FUNCTION_BLOCK BurnOffStation
VAR_INPUT
END_VAR
VAR_OUTPUT
END_VAR
VAR
	HeaterONTimer : TON;
	BlowerOFFTimer : TON;
	PrevRunning, CurrRunning : BOOL := FALSE;
	StartFromReset, StopAfterEStop : BOOL:=FALSE;	
	BlowerEnable: BOOL := FALSE;
	HeatEnable: BOOL := FALSE;
	PIDEnable: BOOL := FALSE;
	nErrorPIDStatus : UINT;
	PIDOutput : LREAL;
	VoltOutReal : LREAL;
	fbBurnoffPID :FB_BasicPID;
	// Temperature needs to be divided by 10 after reading from the TC card
	fProcessValue: LREAL := 0;
END_VAR

fProcessValue := GVL_IO.BU_Temperature/10;	
STATUS.BurnOffTemperature := LREAL_TO_DINT(fProcessValue);

IF (NOT LotsData.Lot.BurnOffEnabled OR STATIONS.fbMMMonitor.IsMMJammed OR Stations.fbCycleControl.StopRequested OR GVL_IO.MachineEStopped OR Status.BurnOffIdle) THEN
	GVL_IO.BU_HeatCntl := 0;
	GVL_IO.BU_BlowCntl := 0;
ELSE 
	// set the blower setpoint from the User configuration in HMI
	GVL_IO.BU_BlowCntl := REAL_TO_INT(CONFIG.BU_BLOWER_SETPOINT/100*32000); 
	IF ( GVL_IO.BU_BlowCntl > 32000) THEN
		GVL_IO.BU_BlowCntl := 32000;
	END_IF
	// set the heater output based on proporational control with limits 
	fbBurnoffPID (fSetpointValue:= LotsData.Lot.BurnOffTemp +25,
					fActualValue := fProcessValue,
					bReset := FALSE,
					fCtrlCycleTime:=TIME_TO_LREAL(T#500MS),
					fKp:=1000,
					fTn:=0,//TIME_TO_LREAL(T#20MS),
					fTv:=0,//TIME_TO_LREAL(T#200MS),
					fTd:=0,//TIME_TO_LREAL(T#100MS),
					fCtrlOutput =>PIDOutput,
					nErrorStatus => nErrorPIDStatus);			
	        
	IF (PIDOutput>32767) THEN
		PIDOutput := 32767; // full heat, a value of  0.5V will be sent to heater control element. We don't want to heater element too hot
	END_IF
	IF (PIDOutput<0) THEN
		PIDOutput := 0; // No heat, a value of 0 V will be sent to heater control element
	END_IF       
		GVL_IO.BU_HeatCntl := LREAL_TO_INT(PIDOutput); // Write this data out to the Analog Output Card
END_IF

AssignStationStatusForHMI();

METHOD PUBLIC AssignStationStatusForHMI : BOOL
VAR_INPUT
END_VAR
Status.StationsState[MM_CONST.BURNOFF_STA_HMI_STATE] := BOOL_TO_INT(HeatEnable);
IF (LotsData.Lot.BurnOffEnabled) THEN
	IF ((ABS(fProcessValue - LotsData.Lot.BurnOffTemp)) > 25) THEN  // to replace with actual setpoint from user screen
    	Status.StationStauts[MM_CONST.BURNOFF_STA_HMI_STATE] := OverallStationStatus.eHoming;
		Status.BurnOffStatusMsg:= 'Not At Temperature!';
		Status.StationInfoString[MM_CONST.BURNOFF_STA_HMI_STATE] := 'Check BurnOff Leister Powered ON';
	ELSE	
		Status.StationStauts[MM_CONST.BURNOFF_STA_HMI_STATE] := OverallStationStatus.eRunning;
		Status.BurnOffStatusMsg := 'At Temperature';
		Status.StationInfoString[MM_CONST.BURNOFF_STA_HMI_STATE] := '';
	END_IF
END_IF
END_METHOD

PROPERTY PUBLIC IsAtTemperature : BOOL
GET
IsAtTemperature := TRUE;//(Status.StationStauts[MM_CONST.BURNOFF_STA_HMI_STATE] = OverallStationStatus.eRunning);
END_GET
SET
END_SET
END_PROPERTY

END_FUNCTION_BLOCK

(* stored: Version 1.1.0.1, ProductVersion 3.1.4022.6
   POU BurnOffStation: Id {13ee2654-f908-4dad-a00a-52723e365b0f}, SpecialFunc None
   Method AssignStationStatusForHMI: Id {c6c32236-a437-48e2-a462-5473689983ce}
   Property IsAtTemperature: Id {d9725ae4-5cbf-4d8e-8a7b-58a289bff5d5}
   Get Get: Id {bbe5bd19-a129-42e2-8f92-618c33c117b4}
   Set Set: Id {35ee03f7-3981-461a-b5a2-7fb5e7251f2d} *)
